// SIMATIC S7-200 SMART project (STEP 7-Micro/WIN SMART), CPU ST40

SYMBOL_TABLE 系统符号
Always_On        SM0.0    // 始终接通
END_SYMBOL_TABLE

SUBROUTINE_BLOCK SBR_0:SBR0
TITLE=子程序注释
VAR_INPUT
Err_bool:BOOL;	// L0.0 打印机故障位
Err_Pos:BOOL;	// L0.1 打印机故障位Pos
Reset_Day:BOOL;	// L0.2 故障计数天复位（每天7：00）
Reset_Week:BOOL;	// L0.3 故障计数周复位（每周日7：00）
Reset_Month:BOOL;	// L0.4 故障计数月复位（每月1日7：00）
Err_Reset_Delay:BYTE;	// LB1 第一次自动复位延时
Delay_EMS_Time:BYTE;	// LB2 复位失败给EMS信号延时
Delay_Safety_Time:DWORD;	// LD3 安全复位时间
END_VAR
VAR_IN_OUT
TI_1:DWORD;	// LD7 计时1
TI_2:DWORD;	// LD11 计时2
Err_OK_Count:DWORD;	// LD15 
END_VAR
VAR_OUTPUT
Err_Time_Min:INT;	// LW19 打印机主机故障持续分钟
Err_Time_Sec:INT;	// LW21 打印机主机故障持续秒
Reset_output:BOOL;	// L23.0 复位输出
Err_To_EMS:BOOL;	// L23.1 故障到EMS
END_VAR
VAR
temp_Delay1:DWORD;	// LD24 
temp_Delay2:DWORD;	// LD28 
temp_Delay3:DWORD;	// LD32 
END_VAR
BEGIN
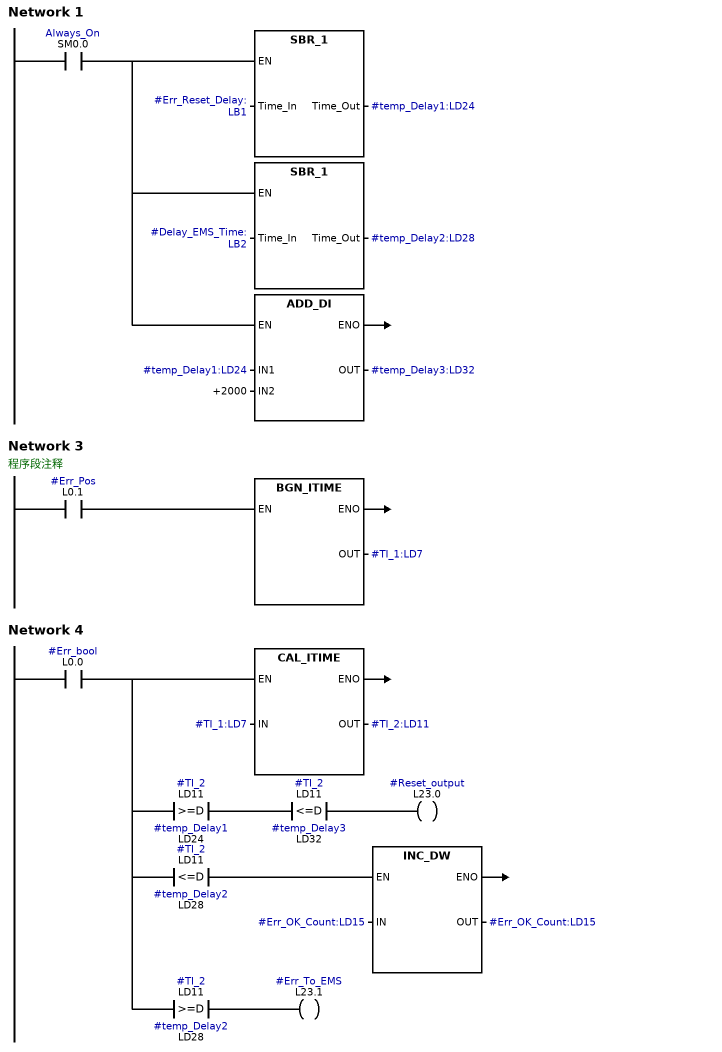
Network 1
// (network saved uncompiled; LAD cells follow)
// row 0: c0 -| |- Always_On:SM0.0 v  c1 --  c2 [SBR_1 EN:=power@row0, Time_In:=#Err_Reset_Delay:LB1, Time_Out=>#temp_Delay1:LD24]
// row 1: c0 ^v  c2 [box]
// row 2: c0 ^v  c1 --  c2 [SBR_1 EN:=power@row2, Time_In:=#Delay_EMS_Time:LB2, Time_Out=>#temp_Delay2:LD28]
// row 3: c0 ^v  c2 [box]
// row 4: c0 ^  c1 --  c2 [ADD_DI EN:=power@row4, IN1:=#temp_Delay1:LD24, IN2:=+2000, ENO=>power, OUT=>#temp_Delay3:LD32]  c3 ->
// row 5: c2 [box]
Network 3
// 程序段注释
LD     #Err_Pos:L0.1
BITIM  #TI_1:LD7
Network 4
// (network saved uncompiled; LAD cells follow)
// row 0: c0 -| |- #Err_bool:L0.0 v  c1 --  c2 [CAL_ITIME EN:=power@row0, IN:=#TI_1:LD7, ENO=>power, OUT=>#TI_2:LD11]  c3 ->
// row 1: c0 ^v  c2 [box]
// row 2: c0 ^v  c1 -|>=D|- #TI_2:LD11, #temp_Delay1:LD24  c2 -|<=D|- #TI_2:LD11, #temp_Delay3:LD32  c3 -( ) #Reset_output:L23.0
// row 3: c0 ^v  c1 -|<=D|- #TI_2:LD11, #temp_Delay2:LD28  c2 --  c3 [INC_DW EN:=power@row3, IN:=#Err_OK_Count:LD15, ENO=>power, OUT=>#Err_OK_Count:LD15]  c4 ->
// row 4: c0 ^v  c3 [box]
// row 5: c0 ^  c1 -|>=D|- #TI_2:LD11, #temp_Delay2:LD28  c2 -( ) #Err_To_EMS:L23.1
END_SUBROUTINE_BLOCK

SUBROUTINE_BLOCK SBR_1:SBR1
TITLE=子程序注释
VAR_INPUT
Time_In:BYTE;	// LB0 
END_VAR
VAR_OUTPUT
Time_Out:DWORD;	// LD1 
END_VAR
VAR
temp1:INT;	// LW5 
temp2:DWORD;	// LD7 
END_VAR
BEGIN
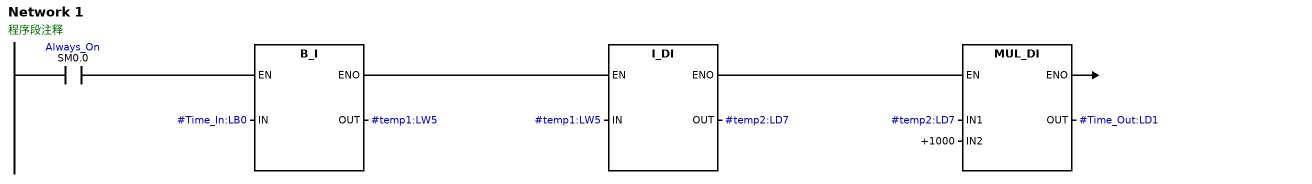
Network 1
// 程序段注释
LD     Always_On:SM0.0
BTI    #Time_In:LB0, #temp1:LW5
AENO
ITD    #temp1:LW5, #temp2:LD7
AENO
MOVD   #temp2:LD7, #Time_Out:LD1
*D     +1000, #Time_Out:LD1
END_SUBROUTINE_BLOCK
